// TIA Portal V15.1 export
// export: Created 2022-03-24T07:02:33.265112Z, ExportSetting WithDefaults, DisplayName Totally Integrated Automation Portal, DisplayVersion V15.1 Update 3, DisplayName TIA Portal Openness, DisplayVersion V15.1, DisplayName TIA Portal Teamcenter Gateway, DisplayVersion V15.1, DisplayName SINAMICS Startdrive Advanced, DisplayVersion V15.1, DisplayName G130, G150, S120, S150, SINAMICS MV, S210, DisplayVersion V15.1, DisplayName G110M, G120, G120C, G120D, G120P, DisplayVersion V15.1, DisplayName STEP 7 Professional, DisplayVersion V15.1 Update 3, DisplayName STEP 7 Safety, DisplayVersion V15.1, DisplayName WinCC Advanced, DisplayVersion V15.1 Update 3
FUNCTION_BLOCK "AS_1390_Typwechsel"   // FB111, GRAPH
{ S7_Optimized_Access := 'TRUE' }
VERSION : 0.1
// stored: AcknowledgeErrorsRequired true, AutoNumber true, GraphVersion 6.0, InitialValuesAcquisition false, IsIECCheckEnabled false, LanguageInNetworks LAD, LockOperatingMode false, PermanentILProcessingInMANMode false, SetENOAutomatically false, SkipSteps false, UDAEnableTagReadback false, WithAlarmHandling true
   // inherited from GRAPH_BASE
   VAR
      OFF_SQ_BASE : Bool;
   END_VAR
   VAR_INPUT
      OFF_SQ { ExternalWritable := 'False'} : Bool := false;   // Kette ausschalten / Turn sequence off / Désactiver le graphe / Disattiva catena / Desactivar cadena / 关闭顺控器
      INIT_SQ { ExternalWritable := 'False'} : Bool := false;   // Kette in Initialzustand versetzen / Set sequence to initial state / Mettre le graphe à l'état initial / Imposta catena nello stato iniziale / Poner cadena en estado inicial / 将顺序设置为初始状态
      ACK_EF { ExternalWritable := 'False'} : Bool := false;   // Alle Fehler und Störungen quittieren / Acknowledge all errors and faults / Acquitter toutes les erreurs et perturbations / Conferma tutti gli errori e le anomalie / Acusar todos los errores y fallos / 确认所有的错误和故障
      S_PREV { ExternalWritable := 'False'} : Bool := false;   // Vorherigen Schritt am Parameter S_NO ausgeben / Output previous step in parameter S_NO / Afficher l'étape précédente dans le paramètre S_NO / Emetti il passo precedente nel parametro S_NO / Mostrar la etapa anterior en el parámetro S_NO / 在S_NO输出参数中显示前导步
      S_NEXT { ExternalWritable := 'False'} : Bool := false;   // Nächsten Schritt am Parameter S_NO anzeigen / Indicate next step in parameter S_NO / Afficher l'étape suivante dans le paramètre S_NO / Visualizza passo successivo nel parametro S_NO / Mostrar la etapa siguiente en el parámetro S_NO / 在S_NO输出参数中显示后续步。
      SW_AUTO { ExternalWritable := 'False'} : Bool := false;   // Automatischer Betrieb / Automatic mode / Mode automatique / Imposta funzionamento automatico / Modo automático / 自动模式
      SW_TAP { ExternalWritable := 'False'} : Bool := false;   // Halbautomatisch/Weiterschalten mit Transition / Semiautomatic/switch with transition / Mode semi-automatique/Activation de l'étape suivante avec transition / Semiautomatico/Avanza con transizione / Semiautomático/continuar con transición / 半自动/转换条件切换
      SW_TOP { ExternalWritable := 'False'} : Bool := false;   // Halbautomatisch/Ignoriere Transition / Semiautomatic/ignore transition / Mode semi-automatique/Ignorer la transition / Semiautomatico/Ignora transizione / Semiautomático/transición ignorada / 半自动/忽略转换条件
      SW_MAN { ExternalWritable := 'False'} : Bool := false;   // Handbetrieb / Manual mode / Mode manuel / Funzionamento manuale / Modo manual / 手动模式
      S_SEL { ExternalWritable := 'False'} : Int := 0;   // Schritt auswählen, der an S_NO ausgegeben werden soll / Select step to be output to S_NO / Sélectionner l'étape à afficher dans S_NO / Seleziona passo da visualizzare in S_NO / Seleccionar la etapa que debe mostrarse en S_NO / 选择要在 S_NO中输出的步。
      S_ON { ExternalWritable := 'False'} : Bool := false;   // Schritt aktivieren, der an Parameter S_NO anliegt / Activate step indicated in S_NO / Activer l'étape figurant dans le paramètre S_NO / Attiva passo visualizzato nel parametro S_NO / Activar la etapa del parámetro S_NO / 激活S_NO 中显示的步。
      S_OFF { ExternalWritable := 'False'} : Bool := false;   // Schritt deaktivieren, der an Parameter S_NO anliegt / Deactivate step indicated S_NO / Désactiver l'étape figurant dans le paramètre S_NO / Disattiva passo visualizzato nel parametro S_NO / Desactivar el incremento presente en el parámetro S_NO / 取消激活 S_NO 中标识的步
      T_PUSH { ExternalWritable := 'False'} : Bool := false;   // Schaltfreigabe für Transition im halbautomatischen Betrieb / Enable transition to switch in semi automatic mode / Validation de commutation pour transition en mode semi-automatique / Abilita commutazione per la transizione nel funzionamento semiautomatico / Habilitar conmutación de transición en modo semiautomático / 允许在半自动模式下跳过转换条件。
   END_VAR
   VAR_OUTPUT
      S_NO { ExternalWritable := 'False'} : Int := 0;   // Schrittnummer / Step number / Numéro d'étape / Numero del passo / Número de etapa / 步编号
      S_MORE { ExternalWritable := 'False'} : Bool := false;   // Weitere Schritte sind vorhanden und können in S_NO angezeigt werden. / More steps are available and can be shown in S_NO / Il existe d'autres étapes qui peuvent être affichées dans S_NO. / Sono presenti altri passi e possono essere visualizzati in S_NO. / Existen más etapas que pueden mostrarse en S_NO. / 更多步可用，并可在S_NO中显示。
      S_ACTIVE { ExternalWritable := 'False'} : Bool := false;   // Schritt, der an Parameter S_NO angezeigt wird, ist aktiv / Step indicated in S_NO is active / L'étape affichée dans le paramètre S_NO est activée / Il passo visualizzato nel parametro S_NO è attivo / El incremento presente en el parámetro S_NO está activo / 在S_NO 中显示的步是激活的。
      ERR_FLT { ExternalWritable := 'False'} : Bool := false;   // Sammelfehler Interlock oder Supervision / Interlock or supervision group error / Erreur groupée Interlock or Supervision / Errore cumulativo interlock o supervisione / Error de grupo interlock o supervisión / 互锁条件或监控条件组出错
      AUTO_ON { ExternalWritable := 'False'} : Bool := false;   // Automatischer Betrieb eingeschaltet / Automatic mode is active / Mode automatique activé / Funzionamento automatico attivo / Modo automático activado / 当前为自动模式
      TAP_ON { ExternalWritable := 'False'} : Bool := false;   // Halbautomatischer Betrieb/Schritt mit Transition eingeschaltet / Semiautomatic mode/step with transition enabled / Mode semi-automatique/Etape avec transition activé / Funzionamento semiautomatico/Passo con transizione attivo / Modo semiautomático/etapa con transición activada / 已启用SW_TAP模式。
      TOP_ON { ExternalWritable := 'False'} : Bool := false;   // Halbautomatischer Betrieb/Ignoriere Transition eingeschaltet / Semiautomatic mode/ignore transition enabled / Mode semi-automatique/Ignorer la transition activé / Semiautomatico/Ignora transizione attivo / Modo semiautomático/Ignorar transición activado / 启用半自动模式/忽略转换条件。
      MAN_ON { ExternalWritable := 'False'} : Bool := false;   // Handbetrieb eingeschaltet / Manual mode is active / Mode manuel activé / Funzionamento manuale attivo / Modo manual activado / 已启用手动模式。
   END_VAR
   VAR_TEMP
      temp : Bool;
   END_VAR
BEGIN
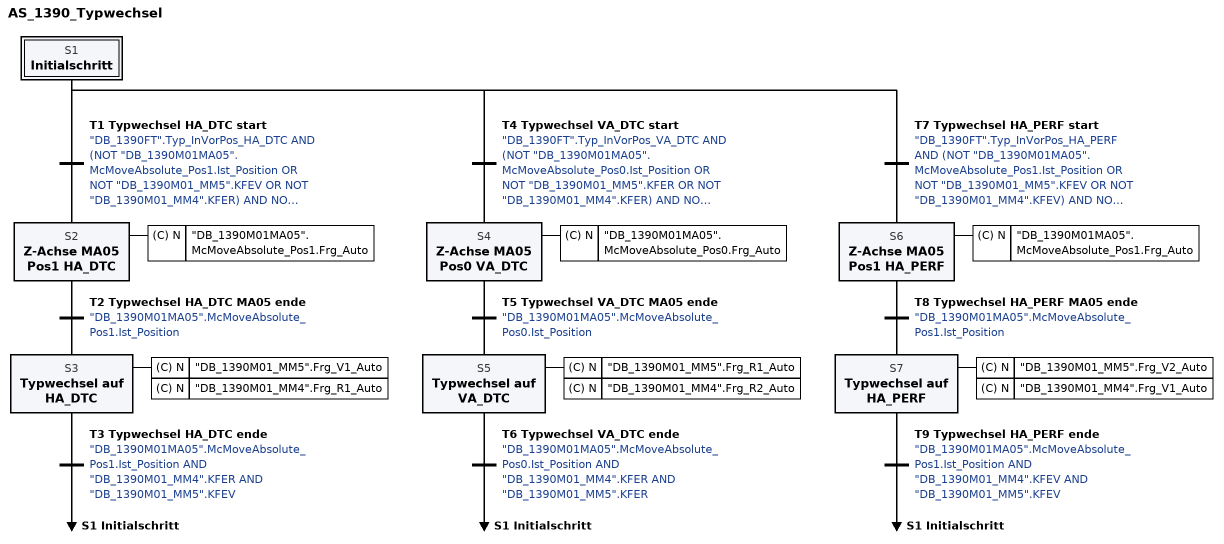
   // sequencer 1: TAF Ablauf
   INITIAL_STEP Initialschritt:   // S1, max time T#10S, warning time T#7S
   END_STEP
   TRANSITION "Typwechsel HA_DTC start" FROM Initialschritt TO "Z-Achse MA05 Pos1 HA_DTC"   // T1
      := "DB_1390FT".Typ_InVorPos_HA_DTC AND (NOT "DB_1390M01MA05".McMoveAbsolute_Pos1.Ist_Position OR NOT "DB_1390M01_MM5".KFEV OR NOT "DB_1390M01_MM4".KFER) AND NOT "DB_1390M01MA130.0".Takt AND "DB_1390FT"."/InPos_MA130.1" AND "DB_1390_BA".PESI;
   END_TRANSITION
   TRANSITION "Typwechsel VA_DTC start" FROM Initialschritt TO "Z-Achse MA05 Pos0 VA_DTC"   // T4
      := "DB_1390FT".Typ_InVorPos_VA_DTC AND (NOT "DB_1390M01MA05".McMoveAbsolute_Pos0.Ist_Position OR NOT "DB_1390M01_MM5".KFER OR NOT "DB_1390M01_MM4".KFER) AND NOT "DB_1390M01MA130.0".Takt AND "DB_1390FT"."/InPos_MA130.1" AND "DB_1390_BA".PESI;
   END_TRANSITION
   TRANSITION "Typwechsel HA_PERF start" FROM Initialschritt TO "Z-Achse MA05 Pos1 HA_PERF"   // T7
      := "DB_1390FT".Typ_InVorPos_HA_PERF AND (NOT "DB_1390M01MA05".McMoveAbsolute_Pos1.Ist_Position OR NOT "DB_1390M01_MM5".KFEV OR NOT "DB_1390M01_MM4".KFEV) AND NOT "DB_1390M01MA130.0".Takt AND "DB_1390FT"."/InPos_MA130.1" AND "DB_1390_BA".PESI;
   END_TRANSITION
   STEP "Z-Achse MA05 Pos1 HA_DTC":   // S2, max time T#10S, warning time T#7S
      interlock C := "DB_1390M01MA04".McMoveAbsolute_Pos0.Ist_Position AND "DB_1390M01MA06".HomePosition AND "DB_1390FT"."/InPos_MA130.1" AND "DB_1390M01_MM1".KFER AND "DB_1390M01_MM2".KFER AND "DB_1390M01_MM3".KFER;
      supervision V := NOT #"Typwechsel HA_DTC MA05 ende".TT AND (#"Z-Achse MA05 Pos1 HA_DTC".U > T#10S);
      (C)     N    "DB_1390M01MA05".McMoveAbsolute_Pos1.Frg_Auto
   END_STEP
   TRANSITION "Typwechsel HA_DTC MA05 ende" FROM "Z-Achse MA05 Pos1 HA_DTC" TO "Typwechsel auf HA_DTC"   // T2
      := "DB_1390M01MA05".McMoveAbsolute_Pos1.Ist_Position;
   END_TRANSITION
   STEP "Typwechsel auf VA_DTC":   // S5, max time T#10S, warning time T#7S
      interlock C := "DB_1390M01MA04".McMoveAbsolute_Pos0.Ist_Position AND "DB_1390M01MA06".HomePosition AND "DB_1390FT"."/InPos_MA130.1" AND "DB_1390M01_MM1".KFER AND "DB_1390M01_MM2".KFER AND "DB_1390M01_MM3".KFER;
      supervision V := NOT #"Typwechsel VA_DTC ende".TT AND (#"Typwechsel auf VA_DTC".U > T#10S);
      (C)     N    "DB_1390M01_MM5".Frg_R1_Auto
      (C)     N    "DB_1390M01_MM4".Frg_R2_Auto
   END_STEP
   TRANSITION "Typwechsel VA_DTC ende" FROM "Typwechsel auf VA_DTC" TO Initialschritt   // T6, jump
      := "DB_1390M01MA05".McMoveAbsolute_Pos0.Ist_Position AND "DB_1390M01_MM4".KFER AND "DB_1390M01_MM5".KFER;
   END_TRANSITION
   STEP "Typwechsel auf HA_PERF":   // S7, max time T#10S, warning time T#7S
      interlock C := "DB_1390M01MA04".McMoveAbsolute_Pos0.Ist_Position AND "DB_1390M01MA06".HomePosition AND "DB_1390FT"."/InPos_MA130.1" AND "DB_1390M01_MM1".KFER AND "DB_1390M01_MM2".KFER AND "DB_1390M01_MM3".KFER;
      supervision V := NOT #"Typwechsel HA_PERF ende".TT AND (#"Typwechsel auf HA_PERF".U > T#10S);
      (C)     N    "DB_1390M01_MM5".Frg_V2_Auto
      (C)     N    "DB_1390M01_MM4".Frg_V1_Auto
   END_STEP
   TRANSITION "Typwechsel HA_PERF ende" FROM "Typwechsel auf HA_PERF" TO Initialschritt   // T9, jump
      := "DB_1390M01MA05".McMoveAbsolute_Pos1.Ist_Position AND "DB_1390M01_MM4".KFEV AND "DB_1390M01_MM5".KFEV;
   END_TRANSITION
   STEP "Typwechsel auf HA_DTC":   // S3, max time T#10S, warning time T#7S
      interlock C := "DB_1390M01MA04".McMoveAbsolute_Pos0.Ist_Position AND "DB_1390M01MA06".HomePosition AND "DB_1390FT"."/InPos_MA130.1" AND "DB_1390M01_MM1".KFER AND "DB_1390M01_MM2".KFER AND "DB_1390M01_MM3".KFER;
      supervision V := NOT #"Typwechsel HA_DTC ende".TT AND (#"Typwechsel auf HA_DTC".U > T#10S);
      (C)     N    "DB_1390M01_MM5".Frg_V1_Auto
      (C)     N    "DB_1390M01_MM4".Frg_R1_Auto
   END_STEP
   TRANSITION "Typwechsel HA_DTC ende" FROM "Typwechsel auf HA_DTC" TO Initialschritt   // T3, jump
      := "DB_1390M01MA05".McMoveAbsolute_Pos1.Ist_Position AND "DB_1390M01_MM4".KFER AND "DB_1390M01_MM5".KFEV;
   END_TRANSITION
   STEP "Z-Achse MA05 Pos0 VA_DTC":   // S4, max time T#10S, warning time T#7S
      interlock C := "DB_1390M01MA04".McMoveAbsolute_Pos0.Ist_Position AND "DB_1390M01MA06".HomePosition AND "DB_1390FT"."/InPos_MA130.1" AND "DB_1390M01_MM1".KFER AND "DB_1390M01_MM2".KFER AND "DB_1390M01_MM3".KFER;
      supervision V := NOT #"Typwechsel VA_DTC MA05 ende".TT AND (#"Z-Achse MA05 Pos0 VA_DTC".U > T#10S);
      (C)     N    "DB_1390M01MA05".McMoveAbsolute_Pos0.Frg_Auto
   END_STEP
   TRANSITION "Typwechsel VA_DTC MA05 ende" FROM "Z-Achse MA05 Pos0 VA_DTC" TO "Typwechsel auf VA_DTC"   // T5
      := "DB_1390M01MA05".McMoveAbsolute_Pos0.Ist_Position;
   END_TRANSITION
   STEP "Z-Achse MA05 Pos1 HA_PERF":   // S6, max time T#10S, warning time T#7S
      interlock C := "DB_1390M01MA04".McMoveAbsolute_Pos0.Ist_Position AND "DB_1390M01MA06".HomePosition AND "DB_1390FT"."/InPos_MA130.1" AND "DB_1390M01_MM1".KFER AND "DB_1390M01_MM2".KFER AND "DB_1390M01_MM3".KFER;
      supervision V := NOT #"Typwechsel HA_PERF MA05 ende".TT AND (#"Z-Achse MA05 Pos1 HA_PERF".U > T#10S);
      (C)     N    "DB_1390M01MA05".McMoveAbsolute_Pos1.Frg_Auto
   END_STEP
   TRANSITION "Typwechsel HA_PERF MA05 ende" FROM "Z-Achse MA05 Pos1 HA_PERF" TO "Typwechsel auf HA_PERF"   // T8
      := "DB_1390M01MA05".McMoveAbsolute_Pos1.Ist_Position;
   END_TRANSITION
END_FUNCTION_BLOCK
